KUKA KRL program: makrosps8.src

&ACCESS RV
&PARAM TEMPLATE = C:\KRC\Roboter\Template\makrospsvorgabe.src
&PARAM EDITMASK = MakroSPS8
&PARAM TPVW_VERSION=8.3.18
DEF MAKROSPS8 ( )
; FOLD Makro Anfang;%{PSE} %MKUKATPVW
SPS_N=-1
; ENDFOLD
; FOLD ;%{H}
END
; ENDFOLD
